(* CODESYS project common.library
   Company: ESO
   Description: This library includes utilities and common structures used by other ESO PLC libraries.
   Version: 0.0.0.1
   Placeholder: ESO LDC Common Library
   Author: Mario Kiekebusch
   Title: ESO LDC Common Library

Project tree, tasks and I/O mapping:
  libraries: Tc2_Standard, * (Beckhoff Automation GmbH); Tc2_System, * (Beckhoff Automation GmbH); Tc3_Module, * (Beckhoff Automation GmbH)
  DUTs/
    Structures/
      data type T_ASTRO_POINTING_KERNEL_POSITIONS
  GVLs/
    global variables GCL
  POUs/
    AstroFunctions/
      function F_Dms2Rad [ST]
      function F_Hms2Rad [ST]
      function F_Rad2Dms [ST]
      function F_Rad2Hms [ST]
      function F_SplitHms [ST]
    NetworkFunctions/
      function F_IpAddress2Integer [ST]
      function F_Integer2IpAddress [ST]
    program MAIN [ST]
  VISUs/
*)

// DUTs/Structures/T_ASTRO_POINTING_KERNEL_POSITIONS
TYPE T_ASTRO_POINTING_KERNEL_POSITIONS :
STRUCT
	target_observed_altaz : 			ARRAY [0..1] OF LREAL;
	current_observed_altaz : 			ARRAY [0..1] OF LREAL;
	time_lst : 							LREAL;
	time_tai : 							LREAL;
	time_utc : 							LREAL;
	north_angle : 						LREAL;
	pupil_angle : 						LREAL;
	elevation_direction_angle : 		LREAL;
	radec_at_altaz_at_requested_xy : 	ARRAY [0..1] OF LREAL;
	observed_altaz_at_requested_xy : 	ARRAY [0..1] OF LREAL;
	parallactic_angle : 				LREAL;
END_STRUCT
END_TYPE

// GVLs/GCL
{attribute 'qualified_only'}
VAR_GLOBAL
	C_PI:				LREAL := 3.1415926535897932384626433832795028841971693993751;
    C_PI2: 				LREAL := C_PI / 2.0;
	C_2PI: 				LREAL := 2.0 * C_PI;
END_VAR

// POUs/AstroFunctions/F_Dms2Rad
(*
 *   astroDms2rad   :   Convert an angle,given in user format, to radians.
 *   ===========
 *
 *   Given    :  angle      an angle as ddmmss.ttt (DegreesMinutesSecs)
 *   Returned :  rad        the angle as radians
 *
 *    The given angle, a floating value in the format DDMMSS.TTT, is 
 *    converted to radians. See also tcsSplitHms.
 *)
FUNCTION F_Dms2Rad : LREAL
VAR_INPUT
	angle:	LREAL;
END_VAR
VAR
	hh,hm,hs:	LREAL;
	ded,der:	LREAL;
END_VAR

(*
double astroDms2rad (double angle)
{
   double hh,hm,hs;
   double ded,der;
   double de2ra = 0.017453292519943;

   astroSplitHms(fabs_(angle),&hh,&hm,&hs);
   ded=hh + hm/60.0 + hs/3600.0;
   if (angle<0.0) ded=-ded; 
   der=ded*de2ra;
   
   return(der);
}*)

F_SplitHms(ABS(angle),h=>hh,m=>hm,sec=>hs);

ded	:= hh + hm/60.0 + hs/3600.0;

IF angle<0.0 THEN
	ded := -ded;
END_IF

der	:= ded * GCL.C_DEG2RAD;


F_Dms2Rad	:= der;

END_FUNCTION

// POUs/AstroFunctions/F_SplitHms
(*
 *   tcsSplitHms   :   Split an angle,given in user format, to its
 *   ===========      parts.
 *
 *   Given    :  angle      an angle as hhmmss.ttt (or ddmmss.tt)
 *   Returned :  h          hours (degrees)
 *               m          minutes (arcminutes)
 *               s          seconds (arcseconds)
 *
 *    The given time/angle, a floating value in the format HHMMSS.TTT, is split
 *    up in the parts HH, MM and SS.TTT (or DDMMSS.TTT if the input parameter
 *    is an angle).  
 *          NOTE:   if the given value is negative, all returned values 
 *    will also be negative! Which is may be not what you want, so take care of
 *    the sign outside of this function!
 * 
 *
 *   EXAMPLES
 *    Example 1:
 *     double time,h,m,s;
 *     time=123456.7;
 *     i=astroSplitHms(time,&h,&m,&s);
 *
 *        will return  h=12.0
 *                     m=34.0
 *                     s=56.7 
 *
 *
 *   Example 2:
 *     double time,h,m,s;
 *     time=345.0;
 *     i=astroSpltHms(time,&h,&m,&s);
 *
 *        will return  h=0.0
 *                     m=3.0
 *                     s=45.0 
 *
 *)
FUNCTION F_SplitHms : bool
VAR_INPUT
	angle:	LREAL;	// an angle as hhmmss.ttt (or ddmmss.tt)
END_VAR
VAR_OUTPUT
	h, m, sec:	LREAL;
END_VAR
VAR
   val:	LREAL;
   hours,minutes,seconds,t1,t2,t3:	LREAL;
 END_VAR

(*
void astroSplitHms (double angle, double *h, double *m, double *s)
{
   double val;
   double hour,min,sec,t1,t2,t3;
   
   val  = angle;  
   sec  = val - (int)(val/100.0)*100.0;    
   t1   = val-sec;
   t2   = t1 - (int)(t1/10000.0)*10000.0;
   min  = t2/100.0;
   t3   = val-sec-t2;
   hour = t3/10000;
   *h   = hour;
   *m   = min;
   *s   = sec;   
   return;
}
*)

val		:= angle;  
seconds	:= val - TRUNC_INT(val/100.0) * 100.0;    
t1		:= val - seconds;
t2		:= t1 - TRUNC_INT(t1/10000.0) * 10000.0;
minutes	:= t2/100.0;
t3		:= val - seconds - t2;
hours	:= t3/10000;

h	:= hours;
m	:= minutes;
sec	:= seconds;   

F_SplitHms	:= TRUE;

END_FUNCTION

// POUs/AstroFunctions/F_Hms2Rad
(*
 *   astroHms2rad   :   Convert a time/angle,given in user format, to radians.
 *   ===========
 *
 *   Given    :  angle      an angle as hhmmss.ttt (HoursMinutesSecs)
 *   Returned :  rad        the angle as radians
 *
 *    The given time/angle, a floating value in the format HHMMSS.TTT, is 
 *    converted to radians. See also tcsSplitHms
 *)
FUNCTION F_Hms2Rad : LREAL
VAR_INPUT
	angle:	LREAL;
END_VAR
VAR
	hh,hm,hs:	LREAL;
	rad,rar:	LREAL;
END_VAR

(*
double astroHms2rad (double angle)
{
   double hh,hm,hs;
   double rad,rar;
   double de2ra = 0.017453292519943;

   astroSplitHms(fabs_(angle),&hh,&hm,&hs);
   rad=(hh + hm/60.0 + hs/3600.0)*15.0;
   rar=rad*de2ra;
   if (angle<0.0) rar=-rar;
   
   return(rar);
}

*)

F_SplitHms(ABS(angle),h=>hh,m=>hm,sec=>hs);

rad	:= (hh + hm/60.0 + hs/3600.0) * 15.0;	// * 15.0 : 24h * 15 = 360 deg
rar	:= rad * GCL.C_DEG2RAD;

IF angle<0.0 THEN
	rar := -rar;
END_IF

F_Hms2Rad	:= rar;

END_FUNCTION

// POUs/AstroFunctions/F_Rad2Dms
FUNCTION F_Rad2Dms : LREAL
VAR_INPUT
	dd:	LREAL;	// angle in radians
END_VAR
VAR
	value:		LREAL;
	degrees:	INT;
	minutes:	INT;
	seconds:	LREAL;
	
	sign:	int := 1;
END_VAR

IF dd < 0.0 THEN
	sign	:= -1;
	dd		:= -dd;
END_IF

value := dd / GCL.C_2PI * 360.0; 	// rad to degrees


degrees	:= TRUNC_INT(value);
minutes := TRUNC_INT((value - degrees)*60.0);
seconds := (value - degrees - minutes/60.0)*3600.0;

					
F_Rad2Dms	:= (degrees * 10000 + minutes * 100 + seconds) * sign;

END_FUNCTION

// POUs/AstroFunctions/F_Rad2Hms
FUNCTION F_Rad2Hms : LREAL
VAR_INPUT
	hh:	LREAL;	// angle in radians
END_VAR
VAR
	value:		LREAL;
	hours:		INT;
	minutes:	INT;
	seconds:	LREAL;
	
	sign:	int := 1;
END_VAR

IF hh < 0.0 THEN
	sign	:= -1;
	hh		:= -hh;
END_IF

value := hh / GCL.C_2PI * 24.0; 	// rad to hours


hours	:= TRUNC_INT(value);
minutes := TRUNC_INT((value - hours)*60.0);
seconds := (value - hours - minutes/60.0)*3600.0;

hours	:= hours * sign;	// put back the sign

					
F_Rad2Hms	:= hours * 10000 + minutes * 100 + seconds;

END_FUNCTION

// POUs/NetworkFunctions/F_IpAddress2Integer
FUNCTION F_IpAddress2Integer : UDINT
VAR_INPUT
	IpAddress : Tc2_System.T_IPv4Addr;
END_VAR
	
VAR
	IpAddressArray : Tc2_System.T_IPv4AddrArr;
    IpAddressInteger : UDINT;
END_VAR

IpAddressArray := Tc2_System.F_ScanIPv4AddrIds(sIPv4 := IpAddress);
IpAddressInteger := LREAL_TO_UDINT(IpAddressArray[0] * EXPT(256, 3) +
                                   IpAddressArray[1] * EXPT(256, 2) +
                                   IpAddressArray[2] * EXPT(256, 1) +
                                   IpAddressArray[3]);

F_IpAddress2Integer := IpAddressInteger;

END_FUNCTION

// POUs/NetworkFunctions/F_Integer2IpAddress
FUNCTION F_Integer2IpAddress : Tc2_System.T_IPv4Addr
VAR_INPUT
	IpAddress : T_IP_ADDRESS;
END_VAR
VAR
	IpAddressArray : Tc2_System.T_IPv4AddrArr;
END_VAR

IpAddressArray[3] := IpAddress.ipAdr[0];
IpAddressArray[2] := IpAddress.ipAdr[1];
IpAddressArray[1] := IpAddress.ipAdr[2];
IpAddressArray[0] := IpAddress.ipAdr[3];

F_Integer2IpAddress := F_CreateIPv4Addr( IpAddressArray );

END_FUNCTION

// POUs/MAIN
PROGRAM MAIN
VAR
END_VAR

END_PROGRAM
